PROGRAM F19_ClearInspectionStatistic
VAR
	fbClearFrontScreenStatistic		:	FB_KPI_ClearFrontScreenStatistic;
	fbClearCameraStatistic			:	FB_KPI_ClearCameraInspection;

(*Basic Statistic**************************************************************)
	fbClearPackAggregationStatistic	:	FB_KPI_ClearInspectionStatistic;
	fbClearOuterAggregationStatistic	:	FB_KPI_ClearInspectionStatistic;
	fbClearCaseAggregationStatistic	:	FB_KPI_ClearInspectionStatistic;

(*Extend Statistic***************************************************************)
	fbClearExtPKStatistic				:	FB_KPI_ClearExtPKStatistic;
	fbClearExtOUTStatistic				:	FB_KPI_ClearExtOUTStatistic;
	fbClearExtCSStatistic				:	FB_KPI_ClearExtCSStatistic;

(****************************************************************************)
	fbClearGeneralStatistic			:	FB_KPI_ClearGeneraStatistic;
END_VAR

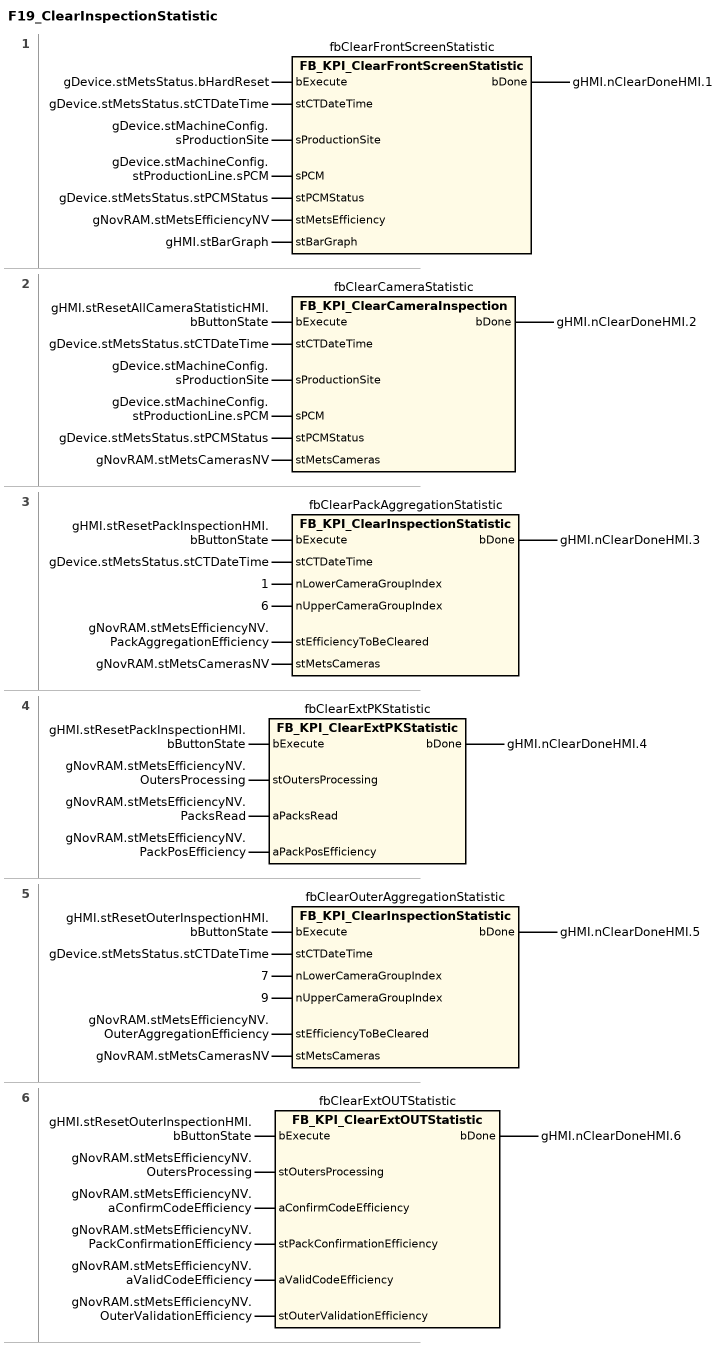
// NETWORK 1
fbClearFrontScreenStatistic(
    bExecute := gDevice.stMetsStatus.bHardReset,
    stCTDateTime := gDevice.stMetsStatus.stCTDateTime,
    sProductionSite := gDevice.stMachineConfig.sProductionSite,
    sPCM := gDevice.stMachineConfig.stProductionLine.sPCM,
    stPCMStatus := gDevice.stMetsStatus.stPCMStatus,
    stMetsEfficiency := gNovRAM.stMetsEfficiencyNV,
    stBarGraph := gHMI.stBarGraph); // FB_KPI_ClearFrontScreenStatistic
gHMI.nClearDoneHMI.1 := fbClearFrontScreenStatistic.bDone;

// NETWORK 2
fbClearCameraStatistic(
    bExecute := gHMI.stResetAllCameraStatisticHMI.bButtonState,
    stCTDateTime := gDevice.stMetsStatus.stCTDateTime,
    sProductionSite := gDevice.stMachineConfig.sProductionSite,
    sPCM := gDevice.stMachineConfig.stProductionLine.sPCM,
    stPCMStatus := gDevice.stMetsStatus.stPCMStatus,
    stMetsCameras := gNovRAM.stMetsCamerasNV); // FB_KPI_ClearCameraInspection
gHMI.nClearDoneHMI.2 := fbClearCameraStatistic.bDone;

// NETWORK 3
fbClearPackAggregationStatistic(
    bExecute := gHMI.stResetPackInspectionHMI.bButtonState,
    stCTDateTime := gDevice.stMetsStatus.stCTDateTime,
    nLowerCameraGroupIndex := 1,
    nUpperCameraGroupIndex := 6,
    stEfficiencyToBeCleared := gNovRAM.stMetsEfficiencyNV.PackAggregationEfficiency,
    stMetsCameras := gNovRAM.stMetsCamerasNV); // FB_KPI_ClearInspectionStatistic
gHMI.nClearDoneHMI.3 := fbClearPackAggregationStatistic.bDone;

// NETWORK 4
fbClearExtPKStatistic(
    bExecute := gHMI.stResetPackInspectionHMI.bButtonState,
    stOutersProcessing := gNovRAM.stMetsEfficiencyNV.OutersProcessing,
    aPacksRead := gNovRAM.stMetsEfficiencyNV.PacksRead,
    aPackPosEfficiency := gNovRAM.stMetsEfficiencyNV.PackPosEfficiency); // FB_KPI_ClearExtPKStatistic
gHMI.nClearDoneHMI.4 := fbClearExtPKStatistic.bDone;

// NETWORK 5
fbClearOuterAggregationStatistic(
    bExecute := gHMI.stResetOuterInspectionHMI.bButtonState,
    stCTDateTime := gDevice.stMetsStatus.stCTDateTime,
    nLowerCameraGroupIndex := 7,
    nUpperCameraGroupIndex := 9,
    stEfficiencyToBeCleared := gNovRAM.stMetsEfficiencyNV.OuterAggregationEfficiency,
    stMetsCameras := gNovRAM.stMetsCamerasNV); // FB_KPI_ClearInspectionStatistic
gHMI.nClearDoneHMI.5 := fbClearOuterAggregationStatistic.bDone;

// NETWORK 6
fbClearExtOUTStatistic(
    bExecute := gHMI.stResetOuterInspectionHMI.bButtonState,
    stOutersProcessing := gNovRAM.stMetsEfficiencyNV.OutersProcessing,
    aConfirmCodeEfficiency := gNovRAM.stMetsEfficiencyNV.aConfirmCodeEfficiency,
    stPackConfirmationEfficiency := gNovRAM.stMetsEfficiencyNV.PackConfirmationEfficiency,
    aValidCodeEfficiency := gNovRAM.stMetsEfficiencyNV.aValidCodeEfficiency,
    stOuterValidationEfficiency := gNovRAM.stMetsEfficiencyNV.OuterValidationEfficiency); // FB_KPI_ClearExtOUTStatistic
gHMI.nClearDoneHMI.6 := fbClearExtOUTStatistic.bDone;

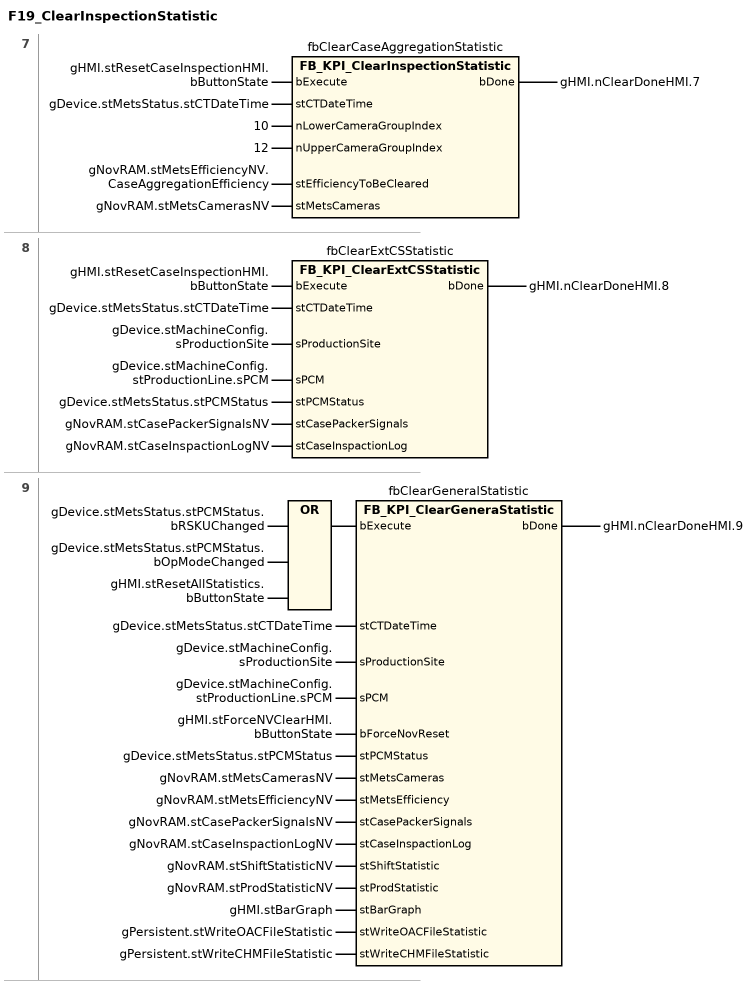
// NETWORK 7
fbClearCaseAggregationStatistic(
    bExecute := gHMI.stResetCaseInspectionHMI.bButtonState,
    stCTDateTime := gDevice.stMetsStatus.stCTDateTime,
    nLowerCameraGroupIndex := 10,
    nUpperCameraGroupIndex := 12,
    stEfficiencyToBeCleared := gNovRAM.stMetsEfficiencyNV.CaseAggregationEfficiency,
    stMetsCameras := gNovRAM.stMetsCamerasNV); // FB_KPI_ClearInspectionStatistic
gHMI.nClearDoneHMI.7 := fbClearCaseAggregationStatistic.bDone;

// NETWORK 8
fbClearExtCSStatistic(
    bExecute := gHMI.stResetCaseInspectionHMI.bButtonState,
    stCTDateTime := gDevice.stMetsStatus.stCTDateTime,
    sProductionSite := gDevice.stMachineConfig.sProductionSite,
    sPCM := gDevice.stMachineConfig.stProductionLine.sPCM,
    stPCMStatus := gDevice.stMetsStatus.stPCMStatus,
    stCasePackerSignals := gNovRAM.stCasePackerSignalsNV,
    stCaseInspactionLog := gNovRAM.stCaseInspactionLogNV); // FB_KPI_ClearExtCSStatistic
gHMI.nClearDoneHMI.8 := fbClearExtCSStatistic.bDone;

// NETWORK 9
fbClearGeneralStatistic(
    bExecute := gDevice.stMetsStatus.stPCMStatus.bRSKUChanged OR gDevice.stMetsStatus.stPCMStatus.bOpModeChanged OR gHMI.stResetAllStatistics.bButtonState,
    stCTDateTime := gDevice.stMetsStatus.stCTDateTime,
    sProductionSite := gDevice.stMachineConfig.sProductionSite,
    sPCM := gDevice.stMachineConfig.stProductionLine.sPCM,
    bForceNovReset := gHMI.stForceNVClearHMI.bButtonState,
    stPCMStatus := gDevice.stMetsStatus.stPCMStatus,
    stMetsCameras := gNovRAM.stMetsCamerasNV,
    stMetsEfficiency := gNovRAM.stMetsEfficiencyNV,
    stCasePackerSignals := gNovRAM.stCasePackerSignalsNV,
    stCaseInspactionLog := gNovRAM.stCaseInspactionLogNV,
    stShiftStatistic := gNovRAM.stShiftStatisticNV,
    stProdStatistic := gNovRAM.stProdStatisticNV,
    stBarGraph := gHMI.stBarGraph,
    stWriteOACFileStatistic := gPersistent.stWriteOACFileStatistic,
    stWriteCHMFileStatistic := gPersistent.stWriteCHMFileStatistic); // FB_KPI_ClearGeneraStatistic
gHMI.nClearDoneHMI.9 := fbClearGeneralStatistic.bDone;

END_PROGRAM

(* stored: Version 1.1.0.1
   POU F19_ClearInspectionStatistic: Id {06714841-db51-4ffb-8642-c65608c7a5bf}, SpecialFunc None *)
